{attribute 'linkalways'} 
{attribute 'no_explicit_call' := 'This FB is a CLASS and must be accessed using methods or properties'}
{attribute 'enable_dynamic_creation'}
FUNCTION_BLOCK _TcVnVector4_INT EXTENDS AliasDatatypeBase
VAR
	localData : TcVnVector4_INT;
	activeData : REFERENCE TO TcVnVector4_INT REF= localData;
	aliasBaseDatatype : _Array0to3OfINT;
END_VAR

PROPERTY PUBLIC Address : PVOID
GET
Address := ADR(activeData);
END_GET
END_PROPERTY

METHOD PUBLIC ClearReference
VAR_INPUT
END_VAR
activeData REF= localData;
SetBaseDatatypeReference();
END_METHOD

METHOD PUBLIC Clone : I_Datatype
VAR
    pClone : POINTER TO _TcVnVector4_INT;
END_VAR
pClone := __NEW(_TcVnVector4_INT);
Clone := pClone^;
END_METHOD

METHOD FB_init : BOOL
VAR_INPUT
	bInitRetains : BOOL; // if TRUE, the retain variables are initialized (warm start / cold start)
	bInCopyCode : BOOL;  // if TRUE, the instance afterwards gets moved into the copy code (online change)
	//InitialValue : <type>; // if possible, not all values can be initialized
END_VAR
//localData := InitialValue; // if possible, not all values can be initialized
SetBaseDatatypeReference();
AddBaseDatatype(aliasBaseDatatype);
END_METHOD

PROPERTY PUBLIC Identifier : T_MAXSTRING
GET
Identifier := 'TcVnVector4_INT';
END_GET
END_PROPERTY

METHOD PUBLIC MakeReferenceTo
VAR_INPUT
	ReferenceTarget : REFERENCE TO TcVnVector4_INT;
END_VAR
activeData REF= ReferenceTarget;
SetBaseDatatypeReference();
END_METHOD

METHOD PROTECTED SetBaseDatatypeReference
VAR_INPUT
END_VAR
aliasBaseDatatype.MakeReferenceTo(activeData);
END_METHOD

PROPERTY PUBLIC Size : UDINT
GET
Size := SIZEOF(activeData);
END_GET
END_PROPERTY

METHOD TryMakeReferenceTo : BOOL
VAR_INPUT
	Target : I_Datatype;
END_VAR
VAR
	pTargetData : POINTER TO TcVnVector4_INT;
END_VAR
IF NOT IsEquivalentTo(Target) THEN
	RETURN;
END_IF

pTargetData := Target.Address;
activeData REF= pTargetData^;
SetBaseDatatypeReference();
TryMakeReferenceTo := TRUE;
END_METHOD

PROPERTY PUBLIC Value : REFERENCE TO TcVnVector4_INT
GET
Value REF= activeData;
END_GET
END_PROPERTY

END_FUNCTION_BLOCK

(* stored: Version 1.1.0.1, ProductVersion 3.1.4024.13
   POU _TcVnVector4_INT: Id {a50c212c-11a1-0751-1dbe-9f74eb094b0e}, SpecialFunc None
   Folder Core: Id {4120e4e7-e3d1-059c-3abc-405d8528526b}
   Folder Protected: Id {ddc74a57-59b5-0b09-0518-8230a6330374}
   Folder Customize: Id {b85120e9-307f-095a-2ebe-c7b3e8141af4}
   Folder Constructor: Id {a90c7ff8-3b1e-0905-2d04-56a6875b00ca}
   Property Address: Id {42542d72-7c94-02d1-349e-ad9b4b819f4b}
   Get Get: Id {0c7bdeb5-2198-0e03-2a6d-449633d88220}
   Method ClearReference: Id {05bcb4e7-6178-08c4-1c99-0462a3ad5939}
   Method Clone: Id {bb70f3b9-b8ec-098c-09af-4e1c77400514}
   Method FB_init: Id {7b355604-8907-040b-3ec4-0aa9ed2a9fa0}
   Property Identifier: Id {f777d702-b53a-06dd-12df-4bbba1b597d7}
   Get Get: Id {c6c5cd2c-befb-0bf2-0ed3-f2bbe75b7530}
   Method MakeReferenceTo: Id {87d501d7-b485-0233-1216-ef63ce96d15c}
   Method SetBaseDatatypeReference: Id {cef8cac4-7d65-0326-2cca-dc45e18ce122}
   Property Size: Id {af1601be-8bf0-033a-1618-2300936d4428}
   Get Get: Id {02424744-eeef-0de0-2fd5-aab4d21d0d61}
   Method TryMakeReferenceTo: Id {4721ded3-0009-0568-3d09-007dac5f9001}
   Property Value: Id {7d814e8b-00f7-0f4c-0482-2cf0a47a4920}
   Get Get: Id {c5919a34-3104-0c79-1608-3dfb09a8547d} *)
